RoboDK station: ImportObj.rdk

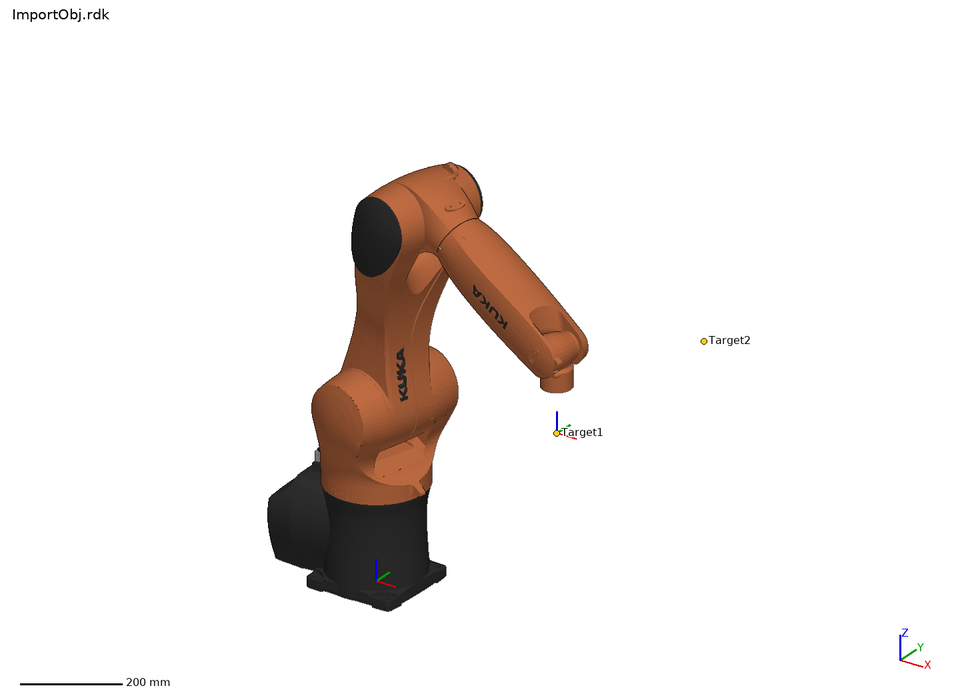
[picture v0: the station drawn from its stored meshes, robots at their saved joint values, targets as dots, program paths as lines]
Station ImportObj (saved by RoboDK 5.4.0). Poses are relative to the parent item; angles as X-Y-Z fixed-axis rotations.
Station parameters (name, value as stored): SizeBox, 123, SizePallet, True, ConvSpeed, True
  - frame RobotBase at (0, 0, 0) mm
    - robot Robot (model KUKA KR 6 R900 sixx): 6 axes, payload 6 kg, reach 901 mm, repeatability 0.03 mm, weight 52 kg
        modified DH rows (alpha deg, a mm, theta deg, d mm): 0, 0, 0, 400; -90, 25, 0, 0; 0, 455, -90, 0; -90, 35, 0, 420; 90, 0, 0, 0; -90, 0, 180, 80
        joint limits [-170, -190, -120, -185, -120, -350] to [170, 45, 156, 185, 120, 350]; home [0, -90, 90, 0, 0, 0]; saved at [11.31, -77.704, 105.45, 180, -62.253, -168.69]
    - target Target1 (Cartesian target) at (500, -100, 500) mm, rotated rx 180 ry 0 rz 180 deg; joints [11.31, -71.252, 112.545, 180, -48.708, -168.69] of Robot
    - target Target2 (Cartesian target) at (500, 400, 500) mm, rotated rx 180 ry 0 rz -180 deg; joints [-38.66, -57.289, 90.823, 0, 56.467, -38.66] of Robot
    - target ChessBoard (Cartesian target) at (500, -100, 500) mm, rotated rx -180 ry 0 rz 180 deg; joints [11.31, -71.252, 112.545, 180, -48.708, -168.69] of Robot
  - frame GlobalZero at (0, 0, 0) mm
  - frame ChessBoard at (500, -100, 500) mm
  - Python program SetParameters (listed below)
  - Python program MoveRobot (listed below)

--- Python program SetParameters ---
# Type help("robolink") or help("robodk") for more information
# Press F5 to run the script
# Note: you do not need to keep a copy of this file, your python script is saved with the station
from robolink import *    # API to communicate with RoboDK
from robodk import *      # basic matrix operations


PARAM_SIZE_BOX = 'SizeBox'
PARAM_SIZE_PALLET = 'SizePallet'
PARAM_CONV_SPEED_MM = 'ConvSpeed'



RDK = Robolink()

size_box = RDK.getParam(PARAM_SIZE_BOX)
size_pallet = RDK.getParam(PARAM_SIZE_PALLET)
conv_speed = RDK.getParam(PARAM_CONV_SPEED_MM)

# ------------------------------------------------------------
size_box_input = mbox('Test', entry=size_box)
if size_box_input:
    RDK.setParam(PARAM_SIZE_BOX, size_box_input)
else:
    raise Exception('Operation cancelled by user')

# ------------------------------------------------------------

--- Python program MoveRobot ---
# Type help("robodk.robolink") or help("robodk.robomath") for more information
# Press F5 to run the script
# Documentation: https://robodk.com/doc/en/RoboDK-API.html
# Reference:     https://robodk.com/doc/en/PythonAPI/index.html
# Note: It is not required to keep a copy of this file, your Python script is saved with your RDK project
from robolink import *    # API to communicate with RoboDK for simulation and offline/online programming
from robodk import *      # Robotics toolbox for industrial robots
from robodk.robomath import *       # import the robotics toolbox


# Any interaction with RoboDK must be done through RDK:
RDK = Robolink()

robot = RDK.Item('Robot', ITEM_TYPE_ROBOT)
target1 = RDK.Item('Target1', ITEM_TYPE_TARGET)
target2 = RDK.Item('Target2', ITEM_TYPE_TARGET)
target3 = RDK.Item('Target3', ITEM_TYPE_TARGET)
ChessBoard = RDK.Item('ChessBoard', ITEM_TYPE_TARGET)
ChessBoardref = RDK.Item('ChessBoard', ITEM_TYPE_FRAME)

robot.setJoints([0,-90,90,0,0,0])   #Set robot to home

robot.MoveJ(target2)
robot.MoveJ(target1)

approach = ChessBoard.Pose()*transl(0,0,-100)
robot.MoveL(approach)
